FUNCTION_BLOCK SlaveAxisPTP EXTENDS AxisPTP IMPLEMENTS I_SlaveAxis
VAR
	// Tasks
	MotionCoupleTaskGearing : MotionCoupleTask_Gearing := (Name := 'MC GearIn Multimaster');
END_VAR

(*FB_Init is always available implicitly and it is used primarily for initialization.
The return value is not evaluated. For a specific influence, you can also declare the
methods explicitly and provide additional code there with the standard initialization
code. You can evaluate the return value.*)
METHOD FB_Init : BOOL
VAR_INPUT
	(* TRUE: the retain variables are initialized (reset warm / reset cold)*)
	bInitRetains : BOOL;

	(* TRUE: the instance will be copied to the copy code afterward (online change)   *)
	bInCopyCode : BOOL;
	Name		: T_MaxString;
	Axis		: REFERENCE TO AXIS_REF;
END_VAR
// Register all Motion Tasks to Collection
MotionTaskCollection.AddTask(MotionCoupleTaskGearing);
END_METHOD

METHOD GearIn
VAR_INPUT
END_VAR
MotionCoupleTaskGearing.GearIn	   := TRUE;
MotionCoupleTaskGearing.BufferMode := _McBufferMode;
MotionCoupleTaskGearing.Execute();
END_METHOD

PROPERTY GearInMultiMasterOptions : ST_GearInMultiMasterOptions
SET
MotionCoupleTaskGearing.GearInMultiMasterOptions := GearInMultiMasterOptions;
END_SET
END_PROPERTY

METHOD GearOut
VAR_INPUT
END_VAR
MotionCoupleTaskGearing.GearIn := FALSE;
MotionCoupleTaskGearing.Execute();
END_METHOD

{attribute 'monitoring' := 'call'}
PROPERTY GearRatioMaster1 : LREAL
SET
MotionCoupleTaskGearing.GearRatioMaster1 := GearRatioMaster1;
END_SET
END_PROPERTY

{attribute 'monitoring' := 'call'}
PROPERTY GearRatioMaster2 : LREAL
SET
MotionCoupleTaskGearing.GearRatioMaster2 := GearRatioMaster2;
END_SET
END_PROPERTY

{attribute 'monitoring' := 'call'}
PROPERTY GearRatioMaster3 : LREAL
SET
MotionCoupleTaskGearing.GearRatioMaster3 := GearRatioMaster3;
END_SET
END_PROPERTY

{attribute 'monitoring' := 'call'}
PROPERTY GearRatioMaster4 : LREAL
SET
MotionCoupleTaskGearing.GearRatioMaster4 := GearRatioMaster4;
END_SET
END_PROPERTY

PROPERTY Master1 : I_Axis
SET
MotionCoupleTaskGearing.Master1 := Master1;
END_SET
END_PROPERTY

PROPERTY Master2 : I_Axis
SET
MotionCoupleTaskGearing.Master2 := Master2;
END_SET
END_PROPERTY

PROPERTY Master3 : I_Axis
SET
MotionCoupleTaskGearing.Master3 := Master3;
END_SET
END_PROPERTY

PROPERTY Master4 : I_Axis
SET
MotionCoupleTaskGearing.Master4 := Master4;
END_SET
END_PROPERTY

END_FUNCTION_BLOCK

(* stored: Version 1.1.0.1, ProductVersion 3.1.4026.18
   POU SlaveAxisPTP: Id {f07e3533-8ef2-4fec-9a40-1320077b46e1}, SpecialFunc None
   Folder Component: Id {fabce388-6807-4b43-b104-1051d8a8e227}
   Folder Slave: Id {25d0cdf1-b946-4279-a4a6-74d6affa85f9}
   Method FB_Init: Id {81ee8f92-5666-41c1-82e5-7ea311e2c2c2}
   Method GearIn: Id {6eec04e7-904d-4015-8412-c0615dca9a2d}
   Property GearInMultiMasterOptions: Id {05b52953-d9ca-42e0-a9b5-0e924f3a1eae}
   Set Set: Id {48563318-c5af-405d-98fd-4981d42d027b}
   Method GearOut: Id {5b215a43-e60f-432c-9737-2f7ad236de4f}
   Property GearRatioMaster1: Id {d82387a1-8184-4a96-bb06-113ac96fe810}
   Set Set: Id {03549ace-b83d-4a99-a836-dcfa422175fa}
   Property GearRatioMaster2: Id {bbef0459-08ad-4663-b5d2-db8a36643387}
   Set Set: Id {ae4f0ce7-bd19-4471-9a61-1e18b7d5b271}
   Property GearRatioMaster3: Id {6c0c7a40-0ccf-43a9-b22a-4dcb7208aedb}
   Set Set: Id {d67e7f6b-6de7-4c46-b097-d1057c93b3fe}
   Property GearRatioMaster4: Id {3c0a6c64-0a0c-4c0a-afb8-1cb3107914fd}
   Set Set: Id {ab86c7c8-0da9-4ad2-9e94-f37c82d956ae}
   Property Master1: Id {2bcfddc7-7c86-42ec-9ead-e61cb9da51c4}
   Set Set: Id {f45f559b-448d-4134-b101-f1c4c1bbf216}
   Property Master2: Id {0b49ac9c-50a2-475e-89d2-711d85e4ec05}
   Set Set: Id {56c94714-3dd4-436d-a21a-e38dc267b7bd}
   Property Master3: Id {4b2cbf9f-3671-4322-95b0-749fb2548772}
   Set Set: Id {3016225c-aed5-41c9-a8bd-e724f583ebc9}
   Property Master4: Id {3b2c84d9-7c7a-470a-a0f2-c6c2c1a9b2f1}
   Set Set: Id {ab99842d-e79a-488d-bdb9-9ba36f591ec5} *)
